Staubli VAL3: onStart.pgx

public program onStart(string& x_sItem[] (dimensions=1))
  local num i
  local string l_sType
begin

end
